// TIA Portal V16 export
// export: Created 2021-07-12T14:47:20.5747506Z, ExportSetting WithDefaults, DisplayName Totally Integrated Automation Portal, DisplayVersion V16, DisplayName TIA Portal Version Control Interface, DisplayVersion V16, DisplayName TIA Portal Openness, DisplayVersion V16, DisplayName STEP 7 Professional, DisplayVersion V16, DisplayName STEP 7 Safety, DisplayVersion V16, DisplayName WinCC Professional, DisplayVersion V16
TYPE "SimaHydTO_typeHMIConnectionGetCharacteristicInterfaceStatus"
TITLE = SimaHydTO_typeHMIConnectionGetCharacteristicInterfaceStatus
// Function block status interface of FB "GetCharacteristics"
// stored: IsFailsafeCompliant false
   STRUCT
      qOutputValueStepForward { ExternalWritable := 'False'} : LReal;   // Last successfully measured manipulated variable in the positive direction
      qOutputValueStepBackward { ExternalWritable := 'False'} : LReal;   // Last successfully measured velocity in the negative direction
      velocityStepForward { ExternalWritable := 'False'} : LReal;   // Last successfully measured velocity in the positive direction
      velocityStepBackward { ExternalWritable := 'False'} : LReal;   // Last successfully measured velocity in the negative direction
      requestForward { ExternalWritable := 'False'} : Bool;   // Request switching to move in the positive direction
      requestBackward { ExternalWritable := 'False'} : Bool;   // Request switching to move in the negative direction
      statusMeasurement { ExternalWritable := 'False'} : Word;   // Status of current measurement
      done { ExternalWritable := 'False'} : Bool;   // The measurement was successfully completed
      busy { ExternalWritable := 'False'} : Bool;   // Measurement active
      commandAborted { ExternalWritable := 'False'} : Bool;   // Measurement function was interrupted
      error { ExternalWritable := 'False'} : Bool;   // There is an error in the FB
      status { ExternalWritable := 'False'} : Word;   // Error information or status of the block
   END_STRUCT;
END_TYPE
